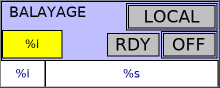
VISUALIZATION VISU_SWEEP_CHEETAH  // 220x88
VAR_IN_OUT
	m_Input_BALAYAGE : BLOCK_TELEMARK_CHEETAH_SWEEP;
END_VAR
    Rectangle (0,0 220x88)
    Rectangle (6,1 117x22), "BALAYAGE"
    Rectangle (0,60 45x27), "%i", text variable: m_Input_BALAYAGE.STATE_NbBal
    Rectangle (45,60 173x27), "%s", text variable: m_Input_BALAYAGE.STATE_BAL
    RoundedRectangle (2,30 60x28), "%i", text variable: m_Input_BALAYAGE.PRM_NbBal, invisible if: NOT Global_Variables.PRG_USER.ACTU_USER.MAINTENANCE OR NOT MACHINE.STATE_Manu, input disabled if: (m_Input_BALAYAGE.STATE_LOC) <> 0
        OnMouseDown: write the text variable via InputWithLimits, min 1, max 8
    RoundedRectangle (163,33 52x23), "ON", invisible if: NOT m_Input_BALAYAGE.STATE_ON
    RoundedRectangle (163,33 52x23), "OFF", invisible if: NOT m_Input_BALAYAGE.STATE_OFF
    RoundedRectangle (128,5 87x23), "REMOTE", invisible if: not m_Input_BALAYAGE.OUT_RMT
    RoundedRectangle (128,5 87x23), "LOCAL", invisible if: m_Input_BALAYAGE.OUT_RMT
    RoundedRectangle (107,33 52x23), "RDY", colour toggle: (m_Input_BALAYAGE.STATE_RDY) <> 0
    Rectangle (126,3 91x27), invisible if: Not m_Input_BALAYAGE.AUTOR_Remote_IHM, input disabled if: NOT PRG_User.ACTU_USER.MAINTENANCE
        tap m_Input_BALAYAGE.M_Remote
    Rectangle (161,31 56x27), invisible if: Not m_Input_BALAYAGE.AUTOR_Balayage_IHM, input disabled if: NOT PRG_User.ACTU_USER.MAINTENANCE
        tap m_Input_BALAYAGE.M_Balayage
END_VISUALIZATION

(* stored: Version 1.1.0.1, ProductVersion 3.1.4026.18
   Visu VISU_SWEEP_CHEETAH: Id {ddbf225d-6238-4cfa-bdd2-3205377efc4a} *)
